GLOBALCONSTANTS AID_EXRN (* External reference name object attribute ids *)
  (* Standard: 61499-1; Description: Copyright (c) 2023 HR Agrartechnik GmbH This program and the accompanying materials are made available under the terms of the Eclipse Public License 2.0 which is available at https://www.eclipse.org/legal/epl-2.0/ SPDX-License-Identifier: EPL-2.0 *)
  (* Version 1.0, 2026-06-20, Franz Höpfinger, HR Agrartechnik GmbH *)
  PACKAGE isobus::UT::Q::const::AID;
  VAR_GLOBAL CONSTANT
    OPTIONS : USINT := USINT#1; (* 1: AID_EXRN_OPTIONS - Bitmask: Bit 0 = Enabled (allows external reference by NAME WS). *)
    NAME_0 : USINT := USINT#2; (* 2: AID_EXRN_NAME_0 *)
    NAME_1 : USINT := USINT#3; (* 3: AID_EXRN_NAME_1 *)
  END_VAR
END_GLOBALCONSTANTS
